FUNCTION_BLOCK M_IO (* Tabular MATRIX I/O *)
  (* Standard: 61499-1; Classification: HMI; Function: MATRIX I/O; Type: Tabular Input *)
  (* Version 0.0, 2002-03-07, JHC, Rockwell Automation *)
  (* Compiler header: package fb.rt.hmi; *)
  (* Compiler Java IBM VisualAge 3.0 *)
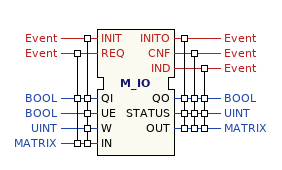
  EVENT_INPUT
    INIT WITH QI, UE, W, IN; (* Initialize matrix to IN *)
    REQ WITH QI, IN; (* Set value to IN *)
  END_EVENT
  EVENT_OUTPUT
    INITO WITH QO, STATUS, OUT; (* Initialization Confirm *)
    CNF WITH QO, STATUS, OUT; (* Confirmation of REQ *)
    IND WITH QO, STATUS, OUT; (* User entered data *)
  END_EVENT
  VAR_INPUT
    QI : BOOL; (* 1=Enabled,0=Inhibited *)
    UE : BOOL; (* 1=Table is User Editable *)
    W : UINT := 10; (* Width of each field in chars *)
    IN : MATRIX; (* Matrix of values to display *)
  END_VAR
  VAR_OUTPUT
    QO : BOOL; (* 0=OK,1=Inhibited *)
    STATUS : UINT; (* 0=OK,2=TYPE_CONVERSION_ERROR,4=INHIBITED,13=ARRAY_SIZE_ERROR *)
    OUT : MATRIX; (* IN value,Possibly User Edited *)
  END_VAR
END_FUNCTION_BLOCK
